TYPE MoveBuffer1kms :
STRUCT
block:	ARRAY[0..1000] OF LREAL;
END_STRUCT
END_TYPE

(* stored: Version 1.1.0.1, ProductVersion 3.1.4024.3
   DUT MoveBuffer1kms: Id {c594af66-502e-404f-b913-83ddcd1f6bc0} *)
